{attribute addProperty BoxType "IL2301-B110-0017"}
{attribute addProperty Id "Term_22KL_5BCCED4C00Term_393_Ix1000KL_9BB4615400"}
{attribute addProperty CRC "3458941263"}
{attribute addProperty SizeInBites "0"}
{attribute addProperty SizeInBytes "0"}
TYPE A_0022_IL2301_B110_0017_CE2B414F EXTENDS IL2301_A5F67C82 :
STRUCT
	{attribute addProperty Name "Term_22"}
	Term_22 : KL_5BCCED4C;
	{attribute addProperty Name "Term_393_Ix1000"}
	Term_393_Ix1000 : KL_9BB46154;
END_STRUCT
END_TYPE

(* stored: Version 1.2.0.0, ProductVersion 3.1.4024.9
   DUT A_0022_IL2301_B110_0017_CE2B414F: Id {de4bfdae-2fd5-44c5-83c5-f9ed5f06d980} *)
